TYPE ST_JntInfo :
STRUCT
	//joint position
	m_curJntPos:LREAL;
	
	//link position
	m_curLinkPos:LREAL;
	
	//Encoder deviation
	m_encErr:LREAL;
	
	//joint maxmum
	m_jntMax:LREAL;
	
	//joint minimum
	m_jntMin:LREAL;
	
	//motor input signal
	m_motorInput:ST_MotorInputs;
	
	//motor output signal
	m_motorOutput:ST_MotorOutputs;
END_STRUCT
END_TYPE

(* stored: Version 1.1.0.1, ProductVersion 3.1.4024.11
   DUT ST_JntInfo: Id {3af648fa-77f6-4329-8684-d0cfd3df649d} *)
